FUNCTION_BLOCK NmGetCfInfoInt (* Service Interface Function Block Type *)
  (* Standard: 61499-2 *)
  (* Version 1.0, 2025-09-04, franz *)
  PACKAGE isobus;
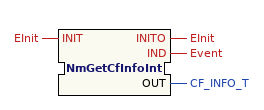
  EVENT_INPUT
    INIT : EInit; (* Service Initialization *)
  END_EVENT
  EVENT_OUTPUT
    INITO : EInit; (* Initialization Confirm *)
    IND; (* Indication from Resource *)
  END_EVENT
  VAR_OUTPUT
    OUT : isobus::pgn::CF_INFO_T;
  END_VAR
END_FUNCTION_BLOCK
